FUNCTION_BLOCK FB_RoutingService_001
VAR_INPUT
	///Calling function number
	eFunctionNumber: E_FunctionNumber;
END_VAR
VAR
	///Debug message service
	fbDebugMsg: FB_DebugMsg;
	///Debug message
	DebugMsg: T_MAXSTRING;
	CurrentZone : ST_ZoneData;
	NextZone : ST_ZoneData;
	TUDest : E_FunctionNumber;
	GetTUIndex233 : DINT;
	GetTUIndex215 : DINT;
	GetTUIndex207 : DINT;
	GetTUIndex232 : DINT;
	GetTUIndex213 : DINT;
	TU_ID : STRING(Conveyor.TU_ID_STRINGLENGTH);
END_VAR
VAR_OUTPUT
	///Result next function number
	eNextFunctionNumber: E_FunctionNumber;
END_VAR


// Example 
// Initialize variable
eNextFunctionNumber := F_BEGIN_FUNCTION;

CASE eFunctionNumber OF
	
	E_FunctionNumber.F_10_001_0200_01_0:
		TUDest := F_PB_GetTuDestination(eFunctionNumber:= eFunctionNumber, 1,1);
		IF TUDest = E_FunctionNumber.F_10_001_0203_01_0 THEN
			eNextFunctionNumber := E_FunctionNumber.F_10_001_0201_01_0;
		END_IF
		
	E_FunctionNumber.F_10_001_0203_01_0:
		NextZone := F_GetZoneData(E_FunctionNumber.F_10_001_0204_01_0, 1);
		IF NOT NextZone.TransportControlData.Occupied THEN
			eNextFunctionNumber := E_FunctionNumber.F_10_001_0204_01_0;
		END_IF
	
	E_FunctionNumber.F_10_001_0204_01_0:
		TUDest := F_PB_GetTuDestination(eFunctionNumber:= eFunctionNumber, 1,1);
		IF TUDest = E_FunctionNumber.F_10_001_0233_01_0 THEN
			eNextFunctionNumber := E_FunctionNumber.F_10_001_0233_01_0;
		ELSE
			eNextFunctionNumber := E_FunctionNumber.F_10_002_0206_01_0;
		END_IF
		
	E_FunctionNumber.F_10_001_0209_01_0:
		TUDest := F_PB_GetTuDestination(eFunctionNumber:= eFunctionNumber, 1,1);
		IF TUDest = E_FunctionNumber.F_10_001_0215_01_0 THEN
			eNextFunctionNumber := E_FunctionNumber.F_10_001_0214_01_0;
		ELSE
			eNextFunctionNumber := E_FunctionNumber.F_10_001_0211_01_0;
		END_IF
		
	E_FunctionNumber.F_10_001_0212_01_0:
		TUDest := F_PB_GetTuDestination(eFunctionNumber:= eFunctionNumber, 1,1);
		NextZone := F_GetZoneData(E_FunctionNumber.F_10_001_0213_01_0, 1);
		IF TUDest = E_FunctionNumber.F_10_001_0213_01_0  AND NOT NextZone.TransportControlData.Occupied THEN
			eNextFunctionNumber := E_FunctionNumber.F_10_001_0213_01_0;
		ELSE
			eNextFunctionNumber := E_FunctionNumber.F_10_001_0218_01_0;
		END_IF
		
	E_FunctionNumber.F_10_001_0222_01_0:
		TUDest := F_PB_GetTuDestination(eFunctionNumber:= eFunctionNumber, 1,1);
		NextZone := F_GetZoneData(E_FunctionNumber.F_10_001_0230_01_0, 1);
		IF (TUDest = E_FunctionNumber.F_10_001_0232_01_0 OR TUDest = E_FunctionNumber.F_10_001_0207_01_0) AND NOT NextZone.TransportControlData.Occupied THEN
			eNextFunctionNumber := E_FunctionNumber.F_10_001_0230_01_0;
		ELSE
			eNextFunctionNumber := E_FunctionNumber.F_10_001_0225_01_0;
		END_IF
		
	E_FunctionNumber.F_10_001_0230_01_0:
		TUDest := F_PB_GetTuDestination(eFunctionNumber:= eFunctionNumber, 1,1);
		IF TUDest = E_FunctionNumber.F_10_001_0232_01_0 THEN
			eNextFunctionNumber := E_FunctionNumber.F_10_001_0232_01_0;
		ELSE
			eNextFunctionNumber := E_FunctionNumber.F_10_001_0207_01_0;
		END_IF
		
		
	// IF position occupied then get data index 
	//When pos not occupied then delete TU data
	E_FunctionNumber.F_10_001_0233_01_0:
		NextZone := F_GetZoneData(E_FunctionNumber.F_10_001_0233_01_0, 1);
		IF NextZone.TransportControlData.Occupied THEN
			GetTUIndex233 := F_GetTU_DataIndex(E_FunctionNumber.F_10_001_0233_01_0, 1);
		ELSE
			F_DeleteTU_Data(GetTUIndex233, FALSE);
			GetTUIndex233 := 0;
		END_IF
	
	E_FunctionNumber.F_10_001_0215_02_0:
		NextZone := F_GetZoneData(E_FunctionNumber.F_10_001_0215_02_0, 1);
		IF NextZone.TransportControlData.Occupied THEN
			GetTUIndex215 := F_GetTU_DataIndex(E_FunctionNumber.F_10_001_0215_02_0, 1);
		ELSE
			F_DeleteTU_Data(GetTUIndex215, FALSE);
			GetTUIndex215 := 0;
		END_IF
		
	E_FunctionNumber.F_10_001_0207_01_0:
		NextZone := F_GetZoneData(E_FunctionNumber.F_10_001_0207_01_0, 1);
		IF NextZone.TransportControlData.Occupied THEN
			GetTUIndex207 := F_GetTU_DataIndex(E_FunctionNumber.F_10_001_0207_01_0, 1);
		ELSE
			F_DeleteTU_Data(GetTUIndex207, FALSE);
			GetTUIndex207 := 0;
		END_IF

	E_FunctionNumber.F_10_001_0232_01_0:
		NextZone := F_GetZoneData(E_FunctionNumber.F_10_001_0232_01_0, 1);
		IF NextZone.TransportControlData.Occupied THEN
			GetTUIndex232 := F_GetTU_DataIndex(E_FunctionNumber.F_10_001_0232_01_0, 1);
		ELSE
			F_DeleteTU_Data(GetTUIndex232, FALSE);
			GetTUIndex232 := 0;
		END_IF
		
	E_FunctionNumber.F_10_001_0213_01_0:
		NextZone := F_GetZoneData(E_FunctionNumber.F_10_001_0213_01_0, 1);
		IF NextZone.TransportControlData.Occupied THEN
			GetTUIndex213 := F_GetTU_DataIndex(E_FunctionNumber.F_10_001_0213_01_0, 1);
		ELSE
			F_DeleteTU_Data(GetTUIndex213, FALSE);
			GetTUIndex213 := 0;
		END_IF
		
	//POR1 an an sis dog schicken von ausgang
	//In sis dog when por1 gekommen schick rtq und tdq
ELSE
	DebugMsg := CONCAT('Routing function not defined. FunctionNumber: ', INT_TO_STRING(eFunctionNumber));
	fbDebugMsg.M_SendInfoMsg(DebugMsg);
END_CASE

END_FUNCTION_BLOCK

(* stored: Version 1.1.0.1, ProductVersion 3.1.4024.9
   POU FB_RoutingService_001: Id {474a0535-b9ae-418c-a013-e57613c2229c}, SpecialFunc None *)
